FUNCTION AxesCalculateTorqueCommandValue : INT
VAR_INPUT
    torqueSetpoint : LREAL; // Nm
    torqueConstant : LREAL; // Nm/A
    channelPeakCurrent : LREAL; // A
END_VAR
VAR
    currentAtMotor : LREAL; // A
    currentFraction : LREAL; // [0.0..1.0]
END_VAR


IF torqueConstant <> 0 THEN
    currentAtMotor := torqueSetpoint / torqueConstant;
ELSE
    currentAtMotor := 0.0;
END_IF

IF channelPeakCurrent <> 0 THEN
    currentFraction := currentAtMotor / channelPeakCurrent;
ELSE
    currentFraction := 0.0;
END_IF

AxesCalculateTorqueCommandValue := LREAL_TO_INT(currentFraction * 1000.0); // units: tenth of a percent ]]>

END_FUNCTION

(* stored: Version 1.1.0.1, ProductVersion 3.1.4018.5
   POU AxesCalculateTorqueCommandValue: Id {fe7fccc7-d63a-478f-bf58-db4847512138}, SpecialFunc None *)
